// TIA Portal project "PLC_Real_programa_proporcional" (V15)

(* hardware
DEVICE "S7-1200 station_1"  S7-1200 Station
   slot 0: "Rack_0"  S7-1200 Rack  Rack  V1.0
   slot 1: "PLC_1"  CPU 1214C DC/DC/DC  6ES7 214-1AE30-0XB0  V2.0
   slot 3: "AQ 1x12BIT_1"  AQ1 signal board  6ES7 232-4HA30-0XB0  V1.0
*)

// ===== PLC "PLC_1"  CPU 1214C DC/DC/DC =====

VAR_GLOBAL   // PLC tag table "Tabla de variables estándar"
   "Valor_Real_Litros" AT %IW64 : Int;
   "Tag_2" AT %QW80 : Int;
   "Marcha" AT %I0.4 : Bool;
   "ON_Variador" AT %Q0.0 : Bool;
   "Sistema_ON" AT %M10.0 : Bool;
   "Paro" AT %I0.3 : Bool;
   "Condicion_1" AT %M20.0 : Bool;
   "Condicion_2" AT %M20.1 : Bool;
   "Condicion_3" AT %M20.2 : Bool;
   "Condicion_4" AT %M20.3 : Bool;
   "Marca_de_simulacion" AT %MW10 : Int;
END_VAR

DATA_BLOCK "Bloque de datos_1"   // DB1
{ S7_Optimized_Access := 'TRUE' }
VERSION : 0.1
   VAR
      ON_Variador : Bool;
      Nivel : Real := 60.0;
      RPM : Real;
   END_VAR
BEGIN
END_DATA_BLOCK

FUNCTION "Acondicionamieno" : Void   // FC1, LAD
{ S7_Optimized_Access := 'TRUE' }
VERSION : 0.1
   VAR_TEMP
      Dato1 : Real;
      Dato2 : Real;
   END_VAR
BEGIN

REGION Network 1
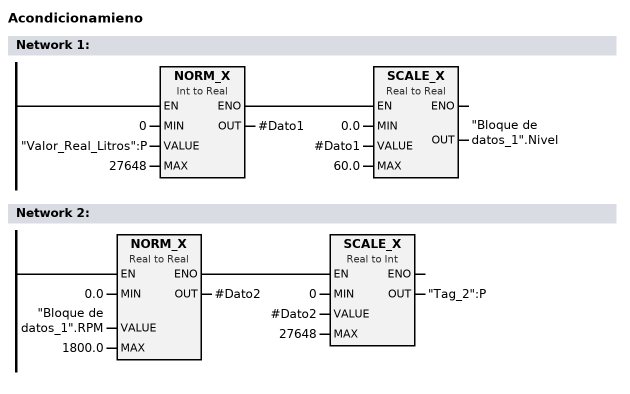
   RUNG wire#powerrail
      { S7_Templates := "[SrcType := Int, DestType := Real]"; S7_GenerateENO := "TRUE" } Normalize(min := 0, value := "Valor_Real_Litros":P, max := 27648, out => #Dato1)
      { S7_Templates := "[SrcType := Real, DestType := Real]"; S7_GenerateENO := "TRUE" } Scale(min := 0.0, value := #Dato1, max := 60.0, out => "Bloque de datos_1".Nivel)
   END_RUNG
   // the same network as SCL:
   // ENO of a box is taken as its EN; it also drops when the box reports an error
   #Dato1 := NORM_X(MIN := 0, VALUE := "Valor_Real_Litros":P, MAX := 27648);
   "Bloque de datos_1".Nivel := SCALE_X(MIN := 0.0, VALUE := #Dato1, MAX := 60.0);
END_REGION

REGION Network 2
   RUNG wire#powerrail
      { S7_Templates := "[SrcType := Real, DestType := Real]"; S7_GenerateENO := "TRUE" } Normalize(min := 0.0, value := "Bloque de datos_1".RPM, max := 1800.0, out => #Dato2)
      { S7_Templates := "[SrcType := Real, DestType := Int]"; S7_GenerateENO := "TRUE" } Scale(min := 0, value := #Dato2, max := 27648, out => "Tag_2":P)
   END_RUNG
   // the same network as SCL:
   // ENO of a box is taken as its EN; it also drops when the box reports an error
   #Dato2 := NORM_X(MIN := 0.0, VALUE := "Bloque de datos_1".RPM, MAX := 1800.0);
   "Tag_2":P := SCALE_X(MIN := 0, VALUE := #Dato2, MAX := 27648);
END_REGION
END_FUNCTION

FUNCTION "Condiciones_de_funcionamiento" : Void   // FC2, LAD
{ S7_Optimized_Access := 'TRUE' }
VERSION : 0.1
BEGIN

REGION Network 1
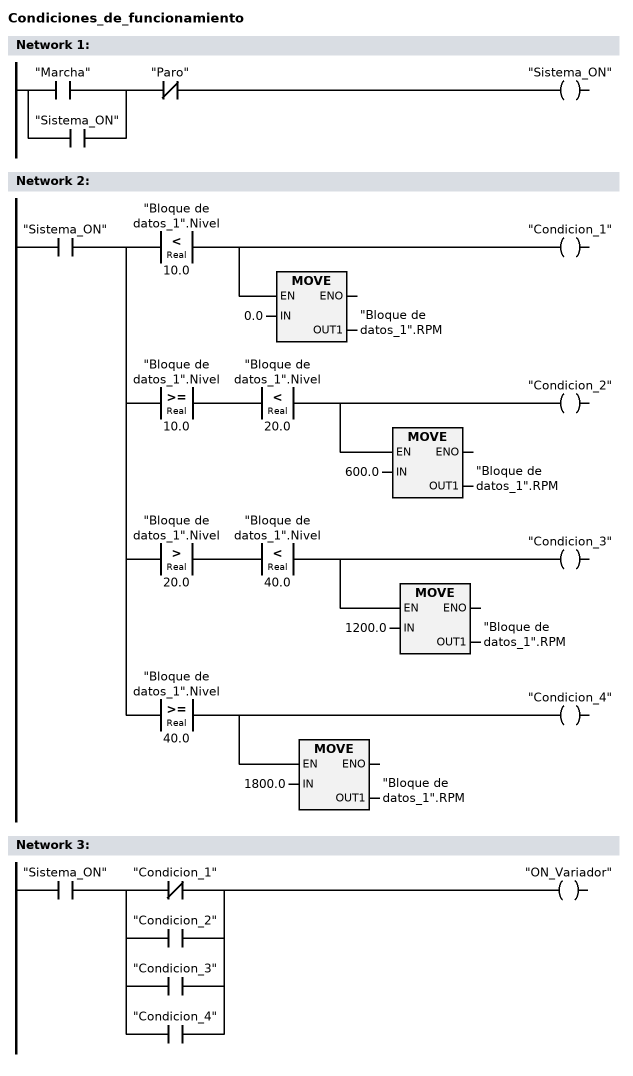
   RUNG wire#powerrail
      Contact( "Marcha" )
      wire#w1
      I_Contact( "Paro" )
      Coil( "Sistema_ON" )
   END_RUNG
   RUNG wire#powerrail
      Contact( "Sistema_ON" )
   END_RUNG wire#w1
   // the same network as SCL:
   "Sistema_ON" := ("Marcha" OR "Sistema_ON") AND NOT "Paro";
END_REGION

REGION Network 2
   RUNG wire#powerrail
      Contact( "Sistema_ON" )
      wire#w1
      { S7_Templates := "SrcType := Real" } LT_Contact(in1 := "Bloque de datos_1".Nivel, in2 := 10.0)
      wire#w2
      Coil( "Condicion_1" )
   END_RUNG
   RUNG wire#w2
      { S7_GenerateENO := "TRUE" } Move(in := 0.0, out1 => "Bloque de datos_1".RPM)
   END_RUNG
   RUNG wire#w1
      { S7_Templates := "SrcType := Real" } GE_Contact(in1 := "Bloque de datos_1".Nivel, in2 := 10.0)
      { S7_Templates := "SrcType := Real" } LT_Contact(in1 := "Bloque de datos_1".Nivel, in2 := 20.0)
      wire#w3
      Coil( "Condicion_2" )
   END_RUNG
   RUNG wire#w3
      { S7_GenerateENO := "TRUE" } Move(in := 600.0, out1 => "Bloque de datos_1".RPM)
   END_RUNG
   RUNG wire#w1
      { S7_Templates := "SrcType := Real" } GT_Contact(in1 := "Bloque de datos_1".Nivel, in2 := 20.0)
      { S7_Templates := "SrcType := Real" } LT_Contact(in1 := "Bloque de datos_1".Nivel, in2 := 40.0)
      wire#w4
      Coil( "Condicion_3" )
   END_RUNG
   RUNG wire#w4
      { S7_GenerateENO := "TRUE" } Move(in := 1200.0, out1 => "Bloque de datos_1".RPM)
   END_RUNG
   RUNG wire#w1
      { S7_Templates := "SrcType := Real" } GE_Contact(in1 := "Bloque de datos_1".Nivel, in2 := 40.0)
      wire#w5
      Coil( "Condicion_4" )
   END_RUNG
   RUNG wire#w5
      { S7_GenerateENO := "TRUE" } Move(in := 1800.0, out1 => "Bloque de datos_1".RPM)
   END_RUNG
   // the same network as SCL:
   "Condicion_1" := "Sistema_ON" AND ("Bloque de datos_1".Nivel < 10.0);
   IF "Condicion_1" THEN "Bloque de datos_1".RPM := 0.0; END_IF;
   "Condicion_2" := "Sistema_ON" AND ("Bloque de datos_1".Nivel >= 10.0) AND ("Bloque de datos_1".Nivel < 20.0);
   IF "Condicion_2" THEN "Bloque de datos_1".RPM := 600.0; END_IF;
   "Condicion_3" := "Sistema_ON" AND ("Bloque de datos_1".Nivel > 20.0) AND ("Bloque de datos_1".Nivel < 40.0);
   IF "Condicion_3" THEN "Bloque de datos_1".RPM := 1200.0; END_IF;
   "Condicion_4" := "Sistema_ON" AND ("Bloque de datos_1".Nivel >= 40.0);
   IF "Condicion_4" THEN "Bloque de datos_1".RPM := 1800.0; END_IF;
END_REGION

REGION Network 3
   RUNG wire#powerrail
      Contact( "Sistema_ON" )
      wire#w1
      I_Contact( "Condicion_1" )
      wire#w2
      Coil( "ON_Variador" )
   END_RUNG
   RUNG wire#w1
      Contact( "Condicion_2" )
   END_RUNG wire#w2
   RUNG wire#w1
      Contact( "Condicion_3" )
   END_RUNG wire#w2
   RUNG wire#w1
      Contact( "Condicion_4" )
   END_RUNG wire#w2
   // the same network as SCL:
   "ON_Variador" := "Sistema_ON" AND (NOT "Condicion_1" OR "Condicion_2" OR "Condicion_3" OR "Condicion_4");
END_REGION
END_FUNCTION

ORGANIZATION_BLOCK "Main"   // OB1, LAD, ProgramCycle
TITLE = "Main Program Sweep (Cycle)"
{ S7_Optimized_Access := 'TRUE' }
VERSION : 0.1
BEGIN

REGION Network 1
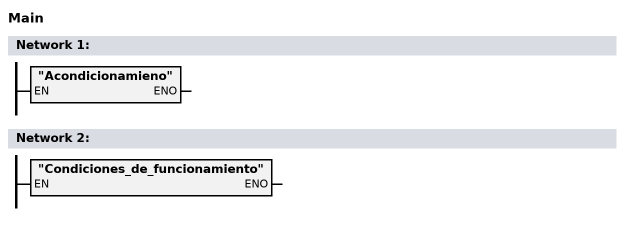
   RUNG wire#powerrail
      "Acondicionamieno"()
   END_RUNG
   // the same network as SCL:
   "Acondicionamieno"();
END_REGION

REGION Network 2
   RUNG wire#powerrail
      "Condiciones_de_funcionamiento"()
   END_RUNG
   // the same network as SCL:
   "Condiciones_de_funcionamiento"();
END_REGION
END_ORGANIZATION_BLOCK